// TIA Portal V16 export
// export: Created 2021-12-01T20:35:58.3632471Z, ExportSetting WithDefaults, DisplayName Totally Integrated Automation Portal, DisplayVersion V16 Update 4, DisplayName TIA Portal Version Control Interface, DisplayVersion V16 Update 2, DisplayName TIA Portal Openness, DisplayVersion V16 Update 4, DisplayName SINAMICS Startdrive Advanced, DisplayVersion V16 Update 5, DisplayName SINAMICS Startdrive G130, G150, S120, S150, SINAMICS MV, S210, DisplayVersion V16 Update 5, DisplayName SINAMICS Startdrive G110M, G120, G120C, G120D, G120P, G115D, DisplayVersion V16 Update 5, DisplayName STEP 7 Professional, DisplayVersion V16 Update 4, DisplayName STEP 7 Safety, DisplayVersion V16, DisplayName WinCC Advanced, DisplayVersion V16 Update 4
FUNCTION "ST00325_FC" : Void   // FC100, LAD
TITLE = ST00325
{ S7_Optimized_Access := 'TRUE' }
VERSION : 0.1
// stored: AutoNumber true, IsIECCheckEnabled false, SetENOAutomatically false, UDAEnableTagReadback false
   VAR_IN_OUT
      OPMODE : "OPMODE_OUT_UDT";
      HMI_EXTENSION : "HMI_EXTENSION_PANEL_UDT";
   END_VAR
   VAR_TEMP
      EmptyHS : "RT_HANDSHAKE_UDT";
      TargetSet : Bool;
      RouteSet : Bool;
      PlantIdentifier : WString;
   END_VAR
   VAR CONSTANT
      SetLocationUID : String := 'ST00325_SL';
      SetPayloadUID : String := 'ST00325_SP';
      SetAttributeUID : String := 'ST00325_SA';
   END_VAR
   VAR_TEMP   // added for the SCL form of the ladder/FBD networks
      _w1 : Bool;
      _w2 : Bool;
   END_VAR
BEGIN

REGION Network 1: Alarm
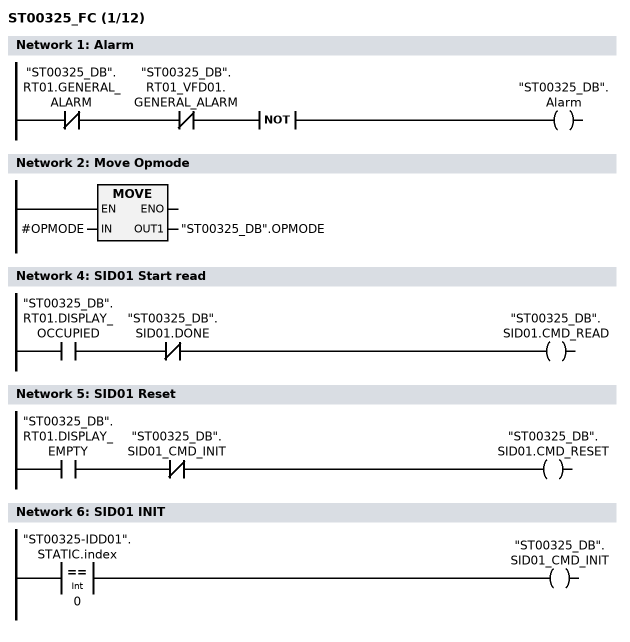
   RUNG wire#powerrail
      I_Contact( "ST00325_DB".RT01.GENERAL_ALARM )
      I_Contact( "ST00325_DB".RT01_VFD01.GENERAL_ALARM )
      Not()
      Coil( "ST00325_DB".Alarm )
   END_RUNG
   // the same network as SCL:
   "ST00325_DB".Alarm := NOT (NOT "ST00325_DB".RT01.GENERAL_ALARM AND NOT "ST00325_DB".RT01_VFD01.GENERAL_ALARM);
END_REGION

REGION Network 2: Move Opmode
   RUNG wire#powerrail
      Move(in := #OPMODE, out1 => "ST00325_DB".OPMODE)
   END_RUNG
   // the same network as SCL:
   "ST00325_DB".OPMODE := #OPMODE;
END_REGION

REGION Network 3: ==== Skid identifier Control ====
END_REGION

REGION Network 4: SID01 Start read
   RUNG wire#powerrail
      Contact( "ST00325_DB".RT01.DISPLAY_OCCUPIED )
      I_Contact( "ST00325_DB".SID01.DONE )
      Coil( "ST00325_DB".SID01.CMD_READ )
   END_RUNG
   // the same network as SCL:
   "ST00325_DB".SID01.CMD_READ := "ST00325_DB".RT01.DISPLAY_OCCUPIED AND NOT "ST00325_DB".SID01.DONE;
END_REGION

REGION Network 5: SID01 Reset
   RUNG wire#powerrail
      Contact( "ST00325_DB".RT01.DISPLAY_EMPTY )
      I_Contact( "ST00325_DB".SID01_CMD_INIT )
      Coil( "ST00325_DB".SID01.CMD_RESET )
   END_RUNG
   // the same network as SCL:
   "ST00325_DB".SID01.CMD_RESET := "ST00325_DB".RT01.DISPLAY_EMPTY AND NOT "ST00325_DB".SID01_CMD_INIT;
END_REGION

REGION Network 6: SID01 INIT
   RUNG wire#powerrail
      { S7_Templates := "SrcType := Int" } EQ_Contact(in1 := "ST00325-IDD01".STATIC.index, in2 := 0)
      Coil( "ST00325_DB".SID01_CMD_INIT )
   END_RUNG
   // the same network as SCL:
   "ST00325_DB".SID01_CMD_INIT := "ST00325-IDD01".STATIC.index = 0;
END_REGION

REGION Network 7: SID01 FB Control
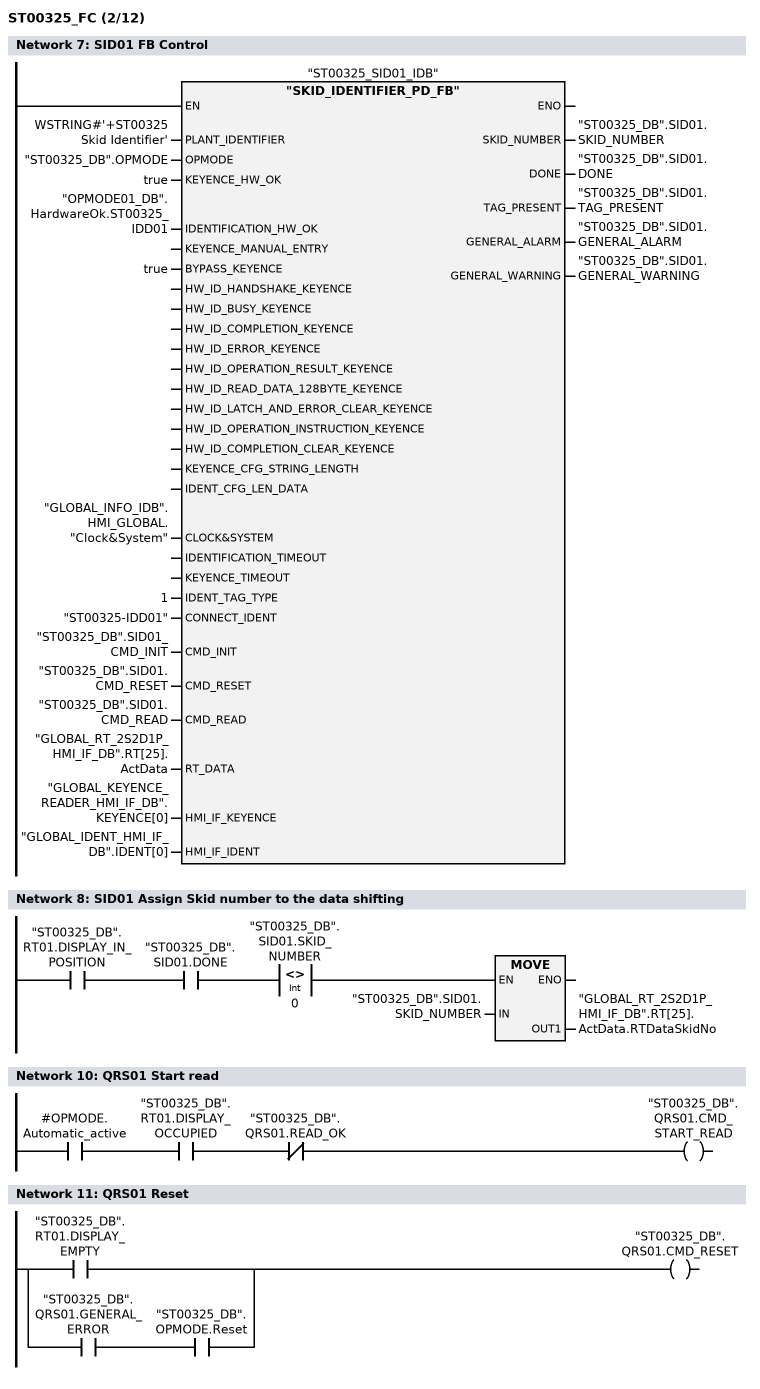
   RUNG wire#powerrail
      "ST00325_SID01_IDB"(PLANT_IDENTIFIER := WSTRING#'+ST00325 Skid Identifier', OPMODE := "ST00325_DB".OPMODE, KEYENCE_HW_OK := true, IDENTIFICATION_HW_OK := "OPMODE01_DB".HardwareOk.ST00325_IDD01, KEYENCE_MANUAL_ENTRY :=, BYPASS_KEYENCE := true, HW_ID_HANDSHAKE_KEYENCE :=, HW_ID_BUSY_KEYENCE :=, HW_ID_COMPLETION_KEYENCE :=, HW_ID_ERROR_KEYENCE :=, HW_ID_OPERATION_RESULT_KEYENCE :=, HW_ID_READ_DATA_128BYTE_KEYENCE :=, HW_ID_LATCH_AND_ERROR_CLEAR_KEYENCE :=, HW_ID_OPERATION_INSTRUCTION_KEYENCE :=, HW_ID_COMPLETION_CLEAR_KEYENCE :=, KEYENCE_CFG_STRING_LENGTH :=, IDENT_CFG_LEN_DATA :=, "CLOCK&SYSTEM" := "GLOBAL_INFO_IDB".HMI_GLOBAL."Clock&System", IDENTIFICATION_TIMEOUT :=, KEYENCE_TIMEOUT :=, IDENT_TAG_TYPE := 1, CONNECT_IDENT := "ST00325-IDD01", CMD_INIT := "ST00325_DB".SID01_CMD_INIT, CMD_RESET := "ST00325_DB".SID01.CMD_RESET, CMD_READ := "ST00325_DB".SID01.CMD_READ, RT_DATA := "GLOBAL_RT_2S2D1P_HMI_IF_DB".RT[25].ActData, HMI_IF_KEYENCE := "GLOBAL_KEYENCE_READER_HMI_IF_DB".KEYENCE[0], HMI_IF_IDENT := "GLOBAL_IDENT_HMI_IF_DB".IDENT[0], SKID_NUMBER => "ST00325_DB".SID01.SKID_NUMBER, DONE => "ST00325_DB".SID01.DONE, TAG_PRESENT => "ST00325_DB".SID01.TAG_PRESENT, GENERAL_ALARM => "ST00325_DB".SID01.GENERAL_ALARM, GENERAL_WARNING => "ST00325_DB".SID01.GENERAL_WARNING)
   END_RUNG
   // the same network as SCL:
   "ST00325_SID01_IDB"(PLANT_IDENTIFIER := WSTRING#'+ST00325 Skid Identifier',   // "SKID_IDENTIFIER_PD_FB"
                       OPMODE := "ST00325_DB".OPMODE,
                       KEYENCE_HW_OK := true,
                       IDENTIFICATION_HW_OK := "OPMODE01_DB".HardwareOk.ST00325_IDD01,
                       BYPASS_KEYENCE := true,
                       "CLOCK&SYSTEM" := "GLOBAL_INFO_IDB".HMI_GLOBAL."Clock&System",
                       IDENT_TAG_TYPE := 1,
                       CONNECT_IDENT := "ST00325-IDD01",
                       CMD_INIT := "ST00325_DB".SID01_CMD_INIT,
                       CMD_RESET := "ST00325_DB".SID01.CMD_RESET,
                       CMD_READ := "ST00325_DB".SID01.CMD_READ,
                       RT_DATA := "GLOBAL_RT_2S2D1P_HMI_IF_DB".RT[25].ActData,
                       HMI_IF_KEYENCE := "GLOBAL_KEYENCE_READER_HMI_IF_DB".KEYENCE[0],
                       HMI_IF_IDENT := "GLOBAL_IDENT_HMI_IF_DB".IDENT[0],
                       SKID_NUMBER => "ST00325_DB".SID01.SKID_NUMBER,
                       DONE => "ST00325_DB".SID01.DONE,
                       TAG_PRESENT => "ST00325_DB".SID01.TAG_PRESENT,
                       GENERAL_ALARM => "ST00325_DB".SID01.GENERAL_ALARM,
                       GENERAL_WARNING => "ST00325_DB".SID01.GENERAL_WARNING);
END_REGION

REGION Network 8: SID01 Assign Skid number to the data shifting
   RUNG wire#powerrail
      Contact( "ST00325_DB".RT01.DISPLAY_IN_POSITION )
      Contact( "ST00325_DB".SID01.DONE )
      { S7_Templates := "SrcType := Int" } NE_Contact(in1 := "ST00325_DB".SID01.SKID_NUMBER, in2 := 0)
      Move(in := "ST00325_DB".SID01.SKID_NUMBER, out1 => "GLOBAL_RT_2S2D1P_HMI_IF_DB".RT[25].ActData.RTDataSkidNo)
   END_RUNG
   // the same network as SCL:
   IF "ST00325_DB".RT01.DISPLAY_IN_POSITION AND "ST00325_DB".SID01.DONE AND ("ST00325_DB".SID01.SKID_NUMBER <> 0) THEN
       "GLOBAL_RT_2S2D1P_HMI_IF_DB".RT[25].ActData.RTDataSkidNo := "ST00325_DB".SID01.SKID_NUMBER;
   END_IF;
END_REGION

REGION Network 9: ==== Camera control ====
END_REGION

REGION Network 10: QRS01 Start read
   RUNG wire#powerrail
      Contact( #OPMODE.Automatic_active )
      Contact( "ST00325_DB".RT01.DISPLAY_OCCUPIED )
      I_Contact( "ST00325_DB".QRS01.READ_OK )
      Coil( "ST00325_DB".QRS01.CMD_START_READ )
   END_RUNG
   // the same network as SCL:
   "ST00325_DB".QRS01.CMD_START_READ := #OPMODE.Automatic_active AND "ST00325_DB".RT01.DISPLAY_OCCUPIED AND NOT "ST00325_DB".QRS01.READ_OK;
END_REGION

REGION Network 11: QRS01 Reset
   RUNG wire#powerrail
      Contact( "ST00325_DB".RT01.DISPLAY_EMPTY )
      wire#w1
      Coil( "ST00325_DB".QRS01.CMD_RESET )
   END_RUNG
   RUNG wire#powerrail
      Contact( "ST00325_DB".QRS01.GENERAL_ERROR )
      Contact( "ST00325_DB".OPMODE.Reset )
   END_RUNG wire#w1
   // the same network as SCL:
   "ST00325_DB".QRS01.CMD_RESET := "ST00325_DB".RT01.DISPLAY_EMPTY OR ("ST00325_DB".QRS01.GENERAL_ERROR AND "ST00325_DB".OPMODE.Reset);
END_REGION

REGION Network 12: QRS01 FB Control
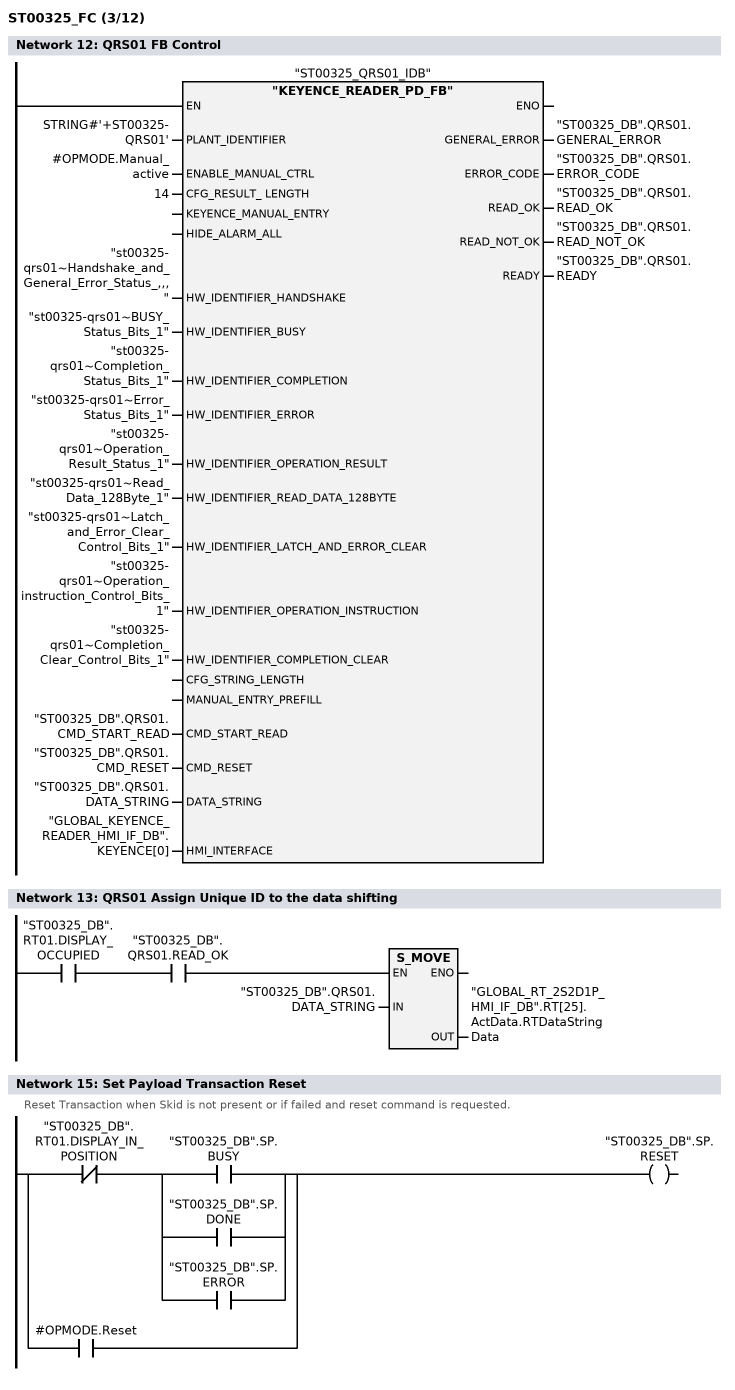
   RUNG wire#powerrail
      "ST00325_QRS01_IDB"(PLANT_IDENTIFIER := STRING#'+ST00325-QRS01', ENABLE_MANUAL_CTRL := #OPMODE.Manual_active, "CFG_RESULT_ LENGTH" := 14, KEYENCE_MANUAL_ENTRY :=, HIDE_ALARM_ALL :=, HW_IDENTIFIER_HANDSHAKE := "st00325-qrs01~Handshake_and_General_Error_Status_,,,", HW_IDENTIFIER_BUSY := "st00325-qrs01~BUSY_Status_Bits_1", HW_IDENTIFIER_COMPLETION := "st00325-qrs01~Completion_Status_Bits_1", HW_IDENTIFIER_ERROR := "st00325-qrs01~Error_Status_Bits_1", HW_IDENTIFIER_OPERATION_RESULT := "st00325-qrs01~Operation_Result_Status_1", HW_IDENTIFIER_READ_DATA_128BYTE := "st00325-qrs01~Read_Data_128Byte_1", HW_IDENTIFIER_LATCH_AND_ERROR_CLEAR := "st00325-qrs01~Latch_and_Error_Clear_Control_Bits_1", HW_IDENTIFIER_OPERATION_INSTRUCTION := "st00325-qrs01~Operation_instruction_Control_Bits_1", HW_IDENTIFIER_COMPLETION_CLEAR := "st00325-qrs01~Completion_Clear_Control_Bits_1", CFG_STRING_LENGTH :=, MANUAL_ENTRY_PREFILL :=, CMD_START_READ := "ST00325_DB".QRS01.CMD_START_READ, CMD_RESET := "ST00325_DB".QRS01.CMD_RESET, DATA_STRING := "ST00325_DB".QRS01.DATA_STRING, HMI_INTERFACE := "GLOBAL_KEYENCE_READER_HMI_IF_DB".KEYENCE[0], GENERAL_ERROR => "ST00325_DB".QRS01.GENERAL_ERROR, ERROR_CODE => "ST00325_DB".QRS01.ERROR_CODE, READ_OK => "ST00325_DB".QRS01.READ_OK, READ_NOT_OK => "ST00325_DB".QRS01.READ_NOT_OK, READY => "ST00325_DB".QRS01.READY)
   END_RUNG
   // the same network as SCL:
   "ST00325_QRS01_IDB"(PLANT_IDENTIFIER := STRING#'+ST00325-QRS01',   // "KEYENCE_READER_PD_FB"
                       ENABLE_MANUAL_CTRL := #OPMODE.Manual_active,
                       "CFG_RESULT_ LENGTH" := 14,
                       HW_IDENTIFIER_HANDSHAKE := "st00325-qrs01~Handshake_and_General_Error_Status_,,,",
                       HW_IDENTIFIER_BUSY := "st00325-qrs01~BUSY_Status_Bits_1",
                       HW_IDENTIFIER_COMPLETION := "st00325-qrs01~Completion_Status_Bits_1",
                       HW_IDENTIFIER_ERROR := "st00325-qrs01~Error_Status_Bits_1",
                       HW_IDENTIFIER_OPERATION_RESULT := "st00325-qrs01~Operation_Result_Status_1",
                       HW_IDENTIFIER_READ_DATA_128BYTE := "st00325-qrs01~Read_Data_128Byte_1",
                       HW_IDENTIFIER_LATCH_AND_ERROR_CLEAR := "st00325-qrs01~Latch_and_Error_Clear_Control_Bits_1",
                       HW_IDENTIFIER_OPERATION_INSTRUCTION := "st00325-qrs01~Operation_instruction_Control_Bits_1",
                       HW_IDENTIFIER_COMPLETION_CLEAR := "st00325-qrs01~Completion_Clear_Control_Bits_1",
                       CMD_START_READ := "ST00325_DB".QRS01.CMD_START_READ,
                       CMD_RESET := "ST00325_DB".QRS01.CMD_RESET,
                       DATA_STRING := "ST00325_DB".QRS01.DATA_STRING,
                       HMI_INTERFACE := "GLOBAL_KEYENCE_READER_HMI_IF_DB".KEYENCE[0],
                       GENERAL_ERROR => "ST00325_DB".QRS01.GENERAL_ERROR,
                       ERROR_CODE => "ST00325_DB".QRS01.ERROR_CODE,
                       READ_OK => "ST00325_DB".QRS01.READ_OK,
                       READ_NOT_OK => "ST00325_DB".QRS01.READ_NOT_OK,
                       READY => "ST00325_DB".QRS01.READY);
END_REGION

REGION Network 13: QRS01 Assign Unique ID to the data shifting
   RUNG wire#powerrail
      Contact( "ST00325_DB".RT01.DISPLAY_OCCUPIED )
      Contact( "ST00325_DB".QRS01.READ_OK )
      S_Move(in := "ST00325_DB".QRS01.DATA_STRING, out => "GLOBAL_RT_2S2D1P_HMI_IF_DB".RT[25].ActData.RTDataStringData)
   END_RUNG
   // the same network as SCL:
   IF "ST00325_DB".RT01.DISPLAY_OCCUPIED AND "ST00325_DB".QRS01.READ_OK THEN
       "GLOBAL_RT_2S2D1P_HMI_IF_DB".RT[25].ActData.RTDataStringData := "ST00325_DB".QRS01.DATA_STRING;
   END_IF;
END_REGION

REGION Network 14: ==== Set Payload ====
   // Set Payload is used to associate a BodyId (payload) to a skid
END_REGION

REGION Network 15: Set Payload Transaction Reset
   // Reset Transaction when Skid is not present or if failed and reset command is requested.
   RUNG wire#powerrail
      I_Contact( "ST00325_DB".RT01.DISPLAY_IN_POSITION )
      wire#w1
      Contact( "ST00325_DB".SP.BUSY )
      wire#w2
      Coil( "ST00325_DB".SP.RESET )
   END_RUNG
   RUNG wire#w1
      Contact( "ST00325_DB".SP.DONE )
   END_RUNG wire#w2
   RUNG wire#w1
      Contact( "ST00325_DB".SP.ERROR )
   END_RUNG wire#w2
   RUNG wire#powerrail
      Contact( #OPMODE.Reset )
   END_RUNG wire#w2
   // the same network as SCL:
   "ST00325_DB".SP.RESET := (NOT "ST00325_DB".RT01.DISPLAY_IN_POSITION AND ("ST00325_DB".SP.BUSY OR "ST00325_DB".SP.DONE OR "ST00325_DB".SP.ERROR)) OR #OPMODE.Reset;
END_REGION

REGION Network 16: Set Payload Transaction Execute
   // Execute Transaction when Skid is present and Skid Number has been retrieved.
   // Prevent further executions if transaction is in progress or has already completed.
   // 
   // To do:
   // - Remove temporary block
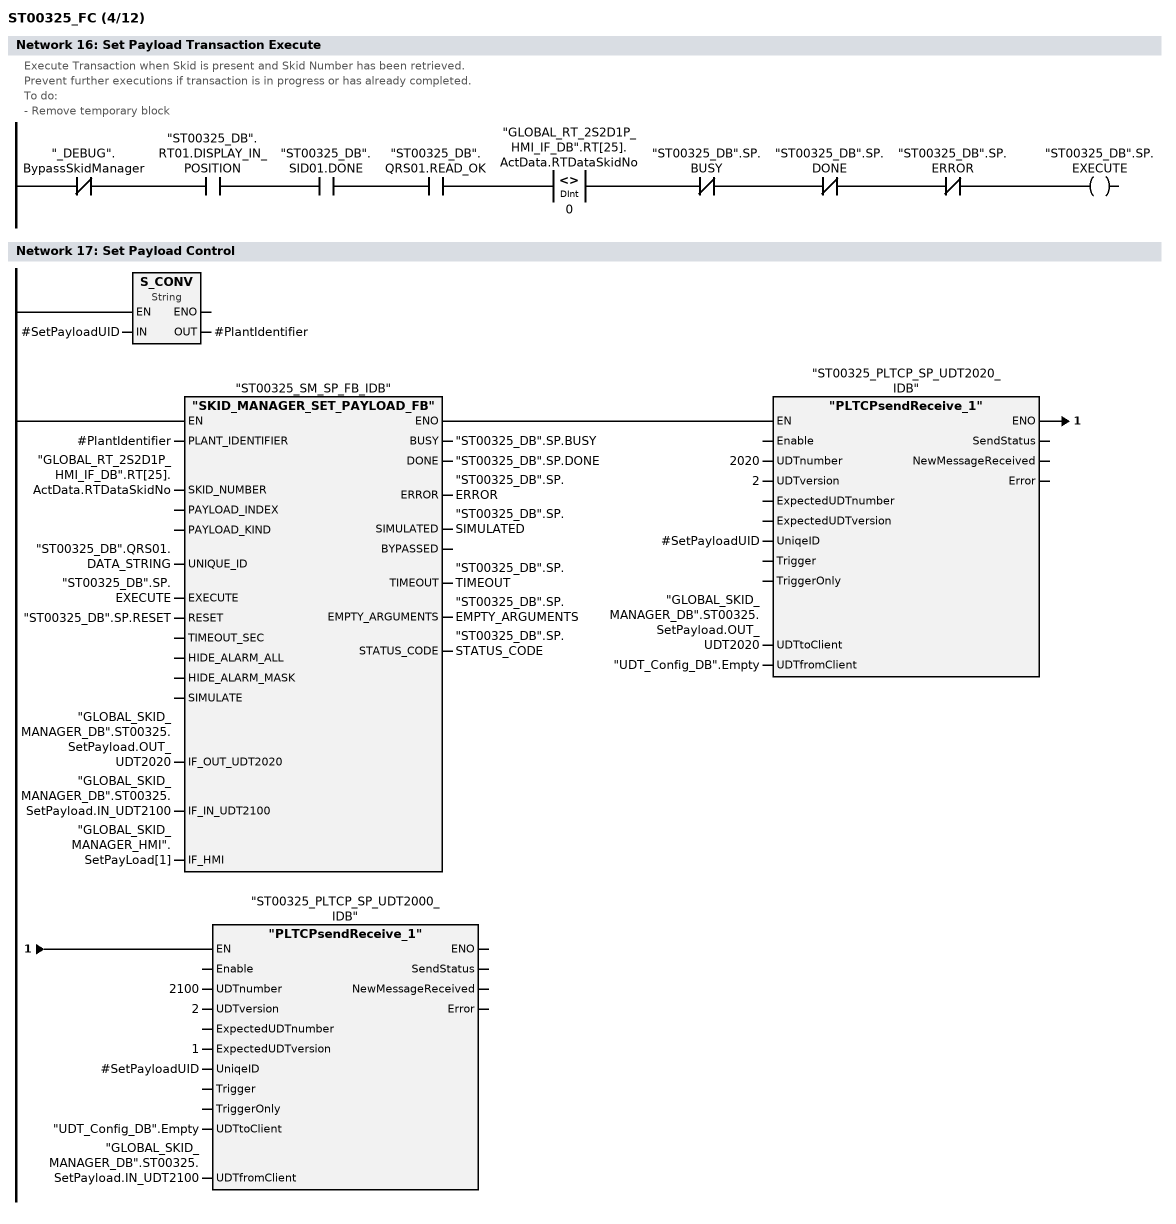
   RUNG wire#powerrail
      I_Contact( "_DEBUG".BypassSkidManager )
      Contact( "ST00325_DB".RT01.DISPLAY_IN_POSITION )
      Contact( "ST00325_DB".SID01.DONE )
      Contact( "ST00325_DB".QRS01.READ_OK )
      { S7_Templates := "SrcType := DInt" } NE_Contact(in1 := "GLOBAL_RT_2S2D1P_HMI_IF_DB".RT[25].ActData.RTDataSkidNo, in2 := 0)
      I_Contact( "ST00325_DB".SP.BUSY )
      I_Contact( "ST00325_DB".SP.DONE )
      I_Contact( "ST00325_DB".SP.ERROR )
      Coil( "ST00325_DB".SP.EXECUTE )
   END_RUNG
   // the same network as SCL:
   "ST00325_DB".SP.EXECUTE := NOT "_DEBUG".BypassSkidManager AND "ST00325_DB".RT01.DISPLAY_IN_POSITION AND "ST00325_DB".SID01.DONE AND "ST00325_DB".QRS01.READ_OK AND ("GLOBAL_RT_2S2D1P_HMI_IF_DB".RT[25].ActData.RTDataSkidNo <> 0) AND NOT "ST00325_DB".SP.BUSY AND NOT "ST00325_DB".SP.DONE AND NOT "ST00325_DB".SP.ERROR;
END_REGION

REGION Network 17: Set Payload Control
   RUNG wire#powerrail
      { S7_Templates := "[src_type := String, dest_type := WString]" } S_CONV(IN := #SetPayloadUID, OUT => #PlantIdentifier)
   END_RUNG
   RUNG wire#powerrail
      "ST00325_SM_SP_FB_IDB"(PLANT_IDENTIFIER := #PlantIdentifier, SKID_NUMBER := "GLOBAL_RT_2S2D1P_HMI_IF_DB".RT[25].ActData.RTDataSkidNo, PAYLOAD_INDEX :=, PAYLOAD_KIND :=, UNIQUE_ID := "ST00325_DB".QRS01.DATA_STRING, EXECUTE := "ST00325_DB".SP.EXECUTE, RESET := "ST00325_DB".SP.RESET, TIMEOUT_SEC :=, HIDE_ALARM_ALL :=, HIDE_ALARM_MASK :=, SIMULATE :=, IF_OUT_UDT2020 := "GLOBAL_SKID_MANAGER_DB".ST00325.SetPayload.OUT_UDT2020, IF_IN_UDT2100 := "GLOBAL_SKID_MANAGER_DB".ST00325.SetPayload.IN_UDT2100, IF_HMI := "GLOBAL_SKID_MANAGER_HMI".SetPayLoad[1], BUSY => "ST00325_DB".SP.BUSY, DONE => "ST00325_DB".SP.DONE, ERROR => "ST00325_DB".SP.ERROR, SIMULATED => "ST00325_DB".SP.SIMULATED, BYPASSED =>, TIMEOUT => "ST00325_DB".SP.TIMEOUT, EMPTY_ARGUMENTS => "ST00325_DB".SP.EMPTY_ARGUMENTS, STATUS_CODE => "ST00325_DB".SP.STATUS_CODE)
      "ST00325_PLTCP_SP_UDT2020_IDB"(Enable :=, UDTnumber := 2020, UDTversion := 2, ExpectedUDTnumber :=, ExpectedUDTversion :=, UniqeID := #SetPayloadUID, Trigger :=, TriggerOnly :=, UDTtoClient := "GLOBAL_SKID_MANAGER_DB".ST00325.SetPayload.OUT_UDT2020, UDTfromClient := "UDT_Config_DB".Empty, SendStatus =>, NewMessageReceived =>, Error =>)
      "ST00325_PLTCP_SP_UDT2000_IDB"(Enable :=, UDTnumber := 2100, UDTversion := 2, ExpectedUDTnumber :=, ExpectedUDTversion := 1, UniqeID := #SetPayloadUID, Trigger :=, TriggerOnly :=, UDTtoClient := "UDT_Config_DB".Empty, UDTfromClient := "GLOBAL_SKID_MANAGER_DB".ST00325.SetPayload.IN_UDT2100, SendStatus =>, NewMessageReceived =>, Error =>)
   END_RUNG
   // the same network as SCL:
   S_CONV(IN := #SetPayloadUID, OUT => #PlantIdentifier);
   "ST00325_SM_SP_FB_IDB"(PLANT_IDENTIFIER := #PlantIdentifier,   // "SKID_MANAGER_SET_PAYLOAD_FB"
                          SKID_NUMBER := "GLOBAL_RT_2S2D1P_HMI_IF_DB".RT[25].ActData.RTDataSkidNo,
                          UNIQUE_ID := "ST00325_DB".QRS01.DATA_STRING,
                          EXECUTE := "ST00325_DB".SP.EXECUTE,
                          RESET := "ST00325_DB".SP.RESET,
                          IF_OUT_UDT2020 := "GLOBAL_SKID_MANAGER_DB".ST00325.SetPayload.OUT_UDT2020,
                          IF_IN_UDT2100 := "GLOBAL_SKID_MANAGER_DB".ST00325.SetPayload.IN_UDT2100,
                          IF_HMI := "GLOBAL_SKID_MANAGER_HMI".SetPayLoad[1],
                          BUSY => "ST00325_DB".SP.BUSY,
                          DONE => "ST00325_DB".SP.DONE,
                          ERROR => "ST00325_DB".SP.ERROR,
                          SIMULATED => "ST00325_DB".SP.SIMULATED,
                          TIMEOUT => "ST00325_DB".SP.TIMEOUT,
                          EMPTY_ARGUMENTS => "ST00325_DB".SP.EMPTY_ARGUMENTS,
                          STATUS_CODE => "ST00325_DB".SP.STATUS_CODE,
                          ENO => #_w1);
   "ST00325_PLTCP_SP_UDT2020_IDB"(EN := #_w1,   // "PLTCPsendReceive_1"
                           UDTnumber := 2020,
                           UDTversion := 2,
                           UniqeID := #SetPayloadUID,
                           UDTtoClient := "GLOBAL_SKID_MANAGER_DB".ST00325.SetPayload.OUT_UDT2020,
                           UDTfromClient := "UDT_Config_DB".Empty,
                           ENO => #_w2);
   IF #_w2 THEN
       "ST00325_PLTCP_SP_UDT2000_IDB"(UDTnumber := 2100,   // "PLTCPsendReceive_1"
                               UDTversion := 2,
                               ExpectedUDTversion := 1,
                               UniqeID := #SetPayloadUID,
                               UDTtoClient := "UDT_Config_DB".Empty,
                               UDTfromClient := "GLOBAL_SKID_MANAGER_DB".ST00325.SetPayload.IN_UDT2100);
   END_IF;
END_REGION

REGION Network 18: ==== Set Location ====
END_REGION

REGION Network 19: Set Location Transaction Reset
   // Reset Transaction when Skid is not present or if failed and reset command is requested.
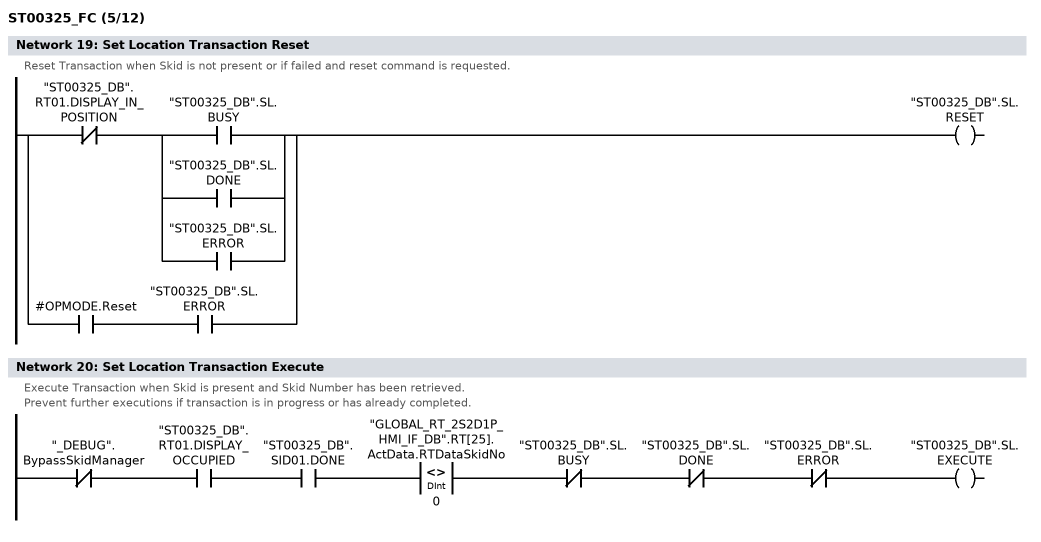
   RUNG wire#powerrail
      I_Contact( "ST00325_DB".RT01.DISPLAY_IN_POSITION )
      wire#w1
      Contact( "ST00325_DB".SL.BUSY )
      wire#w2
      Coil( "ST00325_DB".SL.RESET )
   END_RUNG
   RUNG wire#w1
      Contact( "ST00325_DB".SL.DONE )
   END_RUNG wire#w2
   RUNG wire#w1
      Contact( "ST00325_DB".SL.ERROR )
   END_RUNG wire#w2
   RUNG wire#powerrail
      Contact( #OPMODE.Reset )
      Contact( "ST00325_DB".SL.ERROR )
   END_RUNG wire#w2
   // the same network as SCL:
   "ST00325_DB".SL.RESET := (NOT "ST00325_DB".RT01.DISPLAY_IN_POSITION AND ("ST00325_DB".SL.BUSY OR "ST00325_DB".SL.DONE OR "ST00325_DB".SL.ERROR)) OR (#OPMODE.Reset AND "ST00325_DB".SL.ERROR);
END_REGION

REGION Network 20: Set Location Transaction Execute
   // Execute Transaction when Skid is present and Skid Number has been retrieved.
   // Prevent further executions if transaction is in progress or has already completed.
   RUNG wire#powerrail
      I_Contact( "_DEBUG".BypassSkidManager )
      Contact( "ST00325_DB".RT01.DISPLAY_OCCUPIED )
      Contact( "ST00325_DB".SID01.DONE )
      { S7_Templates := "SrcType := DInt" } NE_Contact(in1 := "GLOBAL_RT_2S2D1P_HMI_IF_DB".RT[25].ActData.RTDataSkidNo, in2 := 0)
      I_Contact( "ST00325_DB".SL.BUSY )
      I_Contact( "ST00325_DB".SL.DONE )
      I_Contact( "ST00325_DB".SL.ERROR )
      Coil( "ST00325_DB".SL.EXECUTE )
   END_RUNG
   // the same network as SCL:
   "ST00325_DB".SL.EXECUTE := NOT "_DEBUG".BypassSkidManager AND "ST00325_DB".RT01.DISPLAY_OCCUPIED AND "ST00325_DB".SID01.DONE AND ("GLOBAL_RT_2S2D1P_HMI_IF_DB".RT[25].ActData.RTDataSkidNo <> 0) AND NOT "ST00325_DB".SL.BUSY AND NOT "ST00325_DB".SL.DONE AND NOT "ST00325_DB".SL.ERROR;
END_REGION

REGION Network 21: Set Location Control
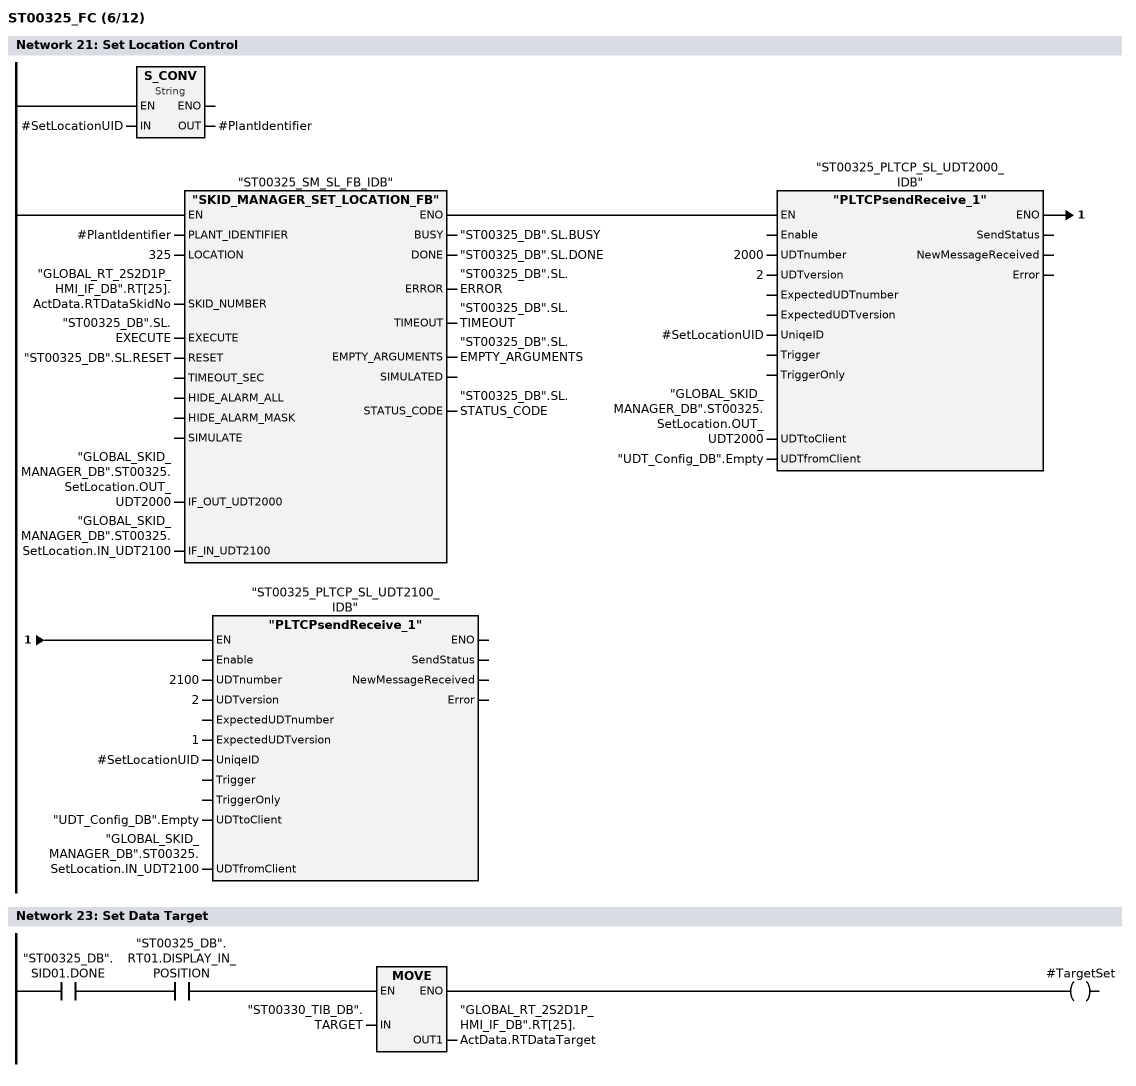
   RUNG wire#powerrail
      { S7_Templates := "[src_type := String, dest_type := WString]" } S_CONV(IN := #SetLocationUID, OUT => #PlantIdentifier)
   END_RUNG
   RUNG wire#powerrail
      "ST00325_SM_SL_FB_IDB"(PLANT_IDENTIFIER := #PlantIdentifier, LOCATION := 325, SKID_NUMBER := "GLOBAL_RT_2S2D1P_HMI_IF_DB".RT[25].ActData.RTDataSkidNo, EXECUTE := "ST00325_DB".SL.EXECUTE, RESET := "ST00325_DB".SL.RESET, TIMEOUT_SEC :=, HIDE_ALARM_ALL :=, HIDE_ALARM_MASK :=, SIMULATE :=, IF_OUT_UDT2000 := "GLOBAL_SKID_MANAGER_DB".ST00325.SetLocation.OUT_UDT2000, IF_IN_UDT2100 := "GLOBAL_SKID_MANAGER_DB".ST00325.SetLocation.IN_UDT2100, BUSY => "ST00325_DB".SL.BUSY, DONE => "ST00325_DB".SL.DONE, ERROR => "ST00325_DB".SL.ERROR, TIMEOUT => "ST00325_DB".SL.TIMEOUT, EMPTY_ARGUMENTS => "ST00325_DB".SL.EMPTY_ARGUMENTS, SIMULATED =>, STATUS_CODE => "ST00325_DB".SL.STATUS_CODE)
      "ST00325_PLTCP_SL_UDT2000_IDB"(Enable :=, UDTnumber := 2000, UDTversion := 2, ExpectedUDTnumber :=, ExpectedUDTversion :=, UniqeID := #SetLocationUID, Trigger :=, TriggerOnly :=, UDTtoClient := "GLOBAL_SKID_MANAGER_DB".ST00325.SetLocation.OUT_UDT2000, UDTfromClient := "UDT_Config_DB".Empty, SendStatus =>, NewMessageReceived =>, Error =>)
      "ST00325_PLTCP_SL_UDT2100_IDB"(Enable :=, UDTnumber := 2100, UDTversion := 2, ExpectedUDTnumber :=, ExpectedUDTversion := 1, UniqeID := #SetLocationUID, Trigger :=, TriggerOnly :=, UDTtoClient := "UDT_Config_DB".Empty, UDTfromClient := "GLOBAL_SKID_MANAGER_DB".ST00325.SetLocation.IN_UDT2100, SendStatus =>, NewMessageReceived =>, Error =>)
   END_RUNG
   // the same network as SCL:
   S_CONV(IN := #SetLocationUID, OUT => #PlantIdentifier);
   "ST00325_SM_SL_FB_IDB"(PLANT_IDENTIFIER := #PlantIdentifier,   // "SKID_MANAGER_SET_LOCATION_FB"
                          LOCATION := 325,
                          SKID_NUMBER := "GLOBAL_RT_2S2D1P_HMI_IF_DB".RT[25].ActData.RTDataSkidNo,
                          EXECUTE := "ST00325_DB".SL.EXECUTE,
                          RESET := "ST00325_DB".SL.RESET,
                          IF_OUT_UDT2000 := "GLOBAL_SKID_MANAGER_DB".ST00325.SetLocation.OUT_UDT2000,
                          IF_IN_UDT2100 := "GLOBAL_SKID_MANAGER_DB".ST00325.SetLocation.IN_UDT2100,
                          BUSY => "ST00325_DB".SL.BUSY,
                          DONE => "ST00325_DB".SL.DONE,
                          ERROR => "ST00325_DB".SL.ERROR,
                          TIMEOUT => "ST00325_DB".SL.TIMEOUT,
                          EMPTY_ARGUMENTS => "ST00325_DB".SL.EMPTY_ARGUMENTS,
                          STATUS_CODE => "ST00325_DB".SL.STATUS_CODE,
                          ENO => #_w1);
   "ST00325_PLTCP_SL_UDT2000_IDB"(EN := #_w1,   // "PLTCPsendReceive_1"
                           UDTnumber := 2000,
                           UDTversion := 2,
                           UniqeID := #SetLocationUID,
                           UDTtoClient := "GLOBAL_SKID_MANAGER_DB".ST00325.SetLocation.OUT_UDT2000,
                           UDTfromClient := "UDT_Config_DB".Empty,
                           ENO => #_w2);
   IF #_w2 THEN
       "ST00325_PLTCP_SL_UDT2100_IDB"(UDTnumber := 2100,   // "PLTCPsendReceive_1"
                               UDTversion := 2,
                               ExpectedUDTversion := 1,
                               UniqeID := #SetLocationUID,
                               UDTtoClient := "UDT_Config_DB".Empty,
                               UDTfromClient := "GLOBAL_SKID_MANAGER_DB".ST00325.SetLocation.IN_UDT2100);
   END_IF;
END_REGION

REGION Network 22: ==== Routing control ====
END_REGION

REGION Network 23: Set Data Target
   RUNG wire#powerrail
      Contact( "ST00325_DB".SID01.DONE )
      Contact( "ST00325_DB".RT01.DISPLAY_IN_POSITION )
      Move(in := "ST00330_TIB_DB".TARGET, out1 => "GLOBAL_RT_2S2D1P_HMI_IF_DB".RT[25].ActData.RTDataTarget)
      Coil( #TargetSet )
   END_RUNG
   // the same network as SCL:
   #_w1 := "ST00325_DB".SID01.DONE AND "ST00325_DB".RT01.DISPLAY_IN_POSITION;
   IF #_w1 THEN "GLOBAL_RT_2S2D1P_HMI_IF_DB".RT[25].ActData.RTDataTarget := "ST00330_TIB_DB".TARGET; END_IF;
   #TargetSet := #_w1;
END_REGION

REGION Network 24: Set route
   // To do:
   // - Determine whether skid is carrying production body or doors/liftgates
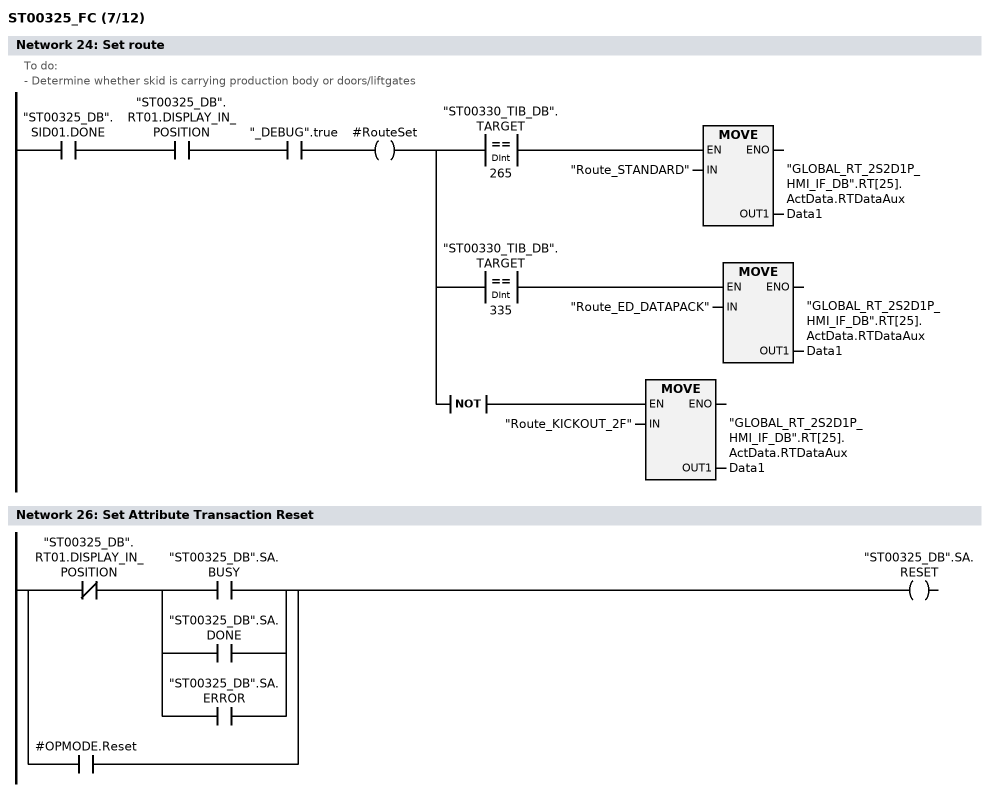
   RUNG wire#powerrail
      Contact( "ST00325_DB".SID01.DONE )
      Contact( "ST00325_DB".RT01.DISPLAY_IN_POSITION )
      Contact( "_DEBUG".true )
      Coil( #RouteSet )
      wire#w1
      { S7_Templates := "SrcType := DInt" } EQ_Contact(in1 := "ST00330_TIB_DB".TARGET, in2 := 265)
      Move(in := "Route_STANDARD", out1 => "GLOBAL_RT_2S2D1P_HMI_IF_DB".RT[25].ActData.RTDataAuxData1)
   END_RUNG
   RUNG wire#w1
      { S7_Templates := "SrcType := DInt" } EQ_Contact(in1 := "ST00330_TIB_DB".TARGET, in2 := 335)
      Move(in := "Route_ED_DATAPACK", out1 => "GLOBAL_RT_2S2D1P_HMI_IF_DB".RT[25].ActData.RTDataAuxData1)
   END_RUNG
   RUNG wire#w1
      Not()
      Move(in := "Route_KICKOUT_2F", out1 => "GLOBAL_RT_2S2D1P_HMI_IF_DB".RT[25].ActData.RTDataAuxData1)
   END_RUNG
   // the same network as SCL:
   #RouteSet := "ST00325_DB".SID01.DONE AND "ST00325_DB".RT01.DISPLAY_IN_POSITION AND "_DEBUG".true;
   IF #RouteSet AND ("ST00330_TIB_DB".TARGET = 265) THEN
       "GLOBAL_RT_2S2D1P_HMI_IF_DB".RT[25].ActData.RTDataAuxData1 := "Route_STANDARD";
   END_IF;
   IF #RouteSet AND ("ST00330_TIB_DB".TARGET = 335) THEN
       "GLOBAL_RT_2S2D1P_HMI_IF_DB".RT[25].ActData.RTDataAuxData1 := "Route_ED_DATAPACK";
   END_IF;
   IF NOT #RouteSet THEN
       "GLOBAL_RT_2S2D1P_HMI_IF_DB".RT[25].ActData.RTDataAuxData1 := "Route_KICKOUT_2F";
   END_IF;
END_REGION

REGION Network 25: ==== Set Attribute ====
END_REGION

REGION Network 26: Set Attribute Transaction Reset
   RUNG wire#powerrail
      I_Contact( "ST00325_DB".RT01.DISPLAY_IN_POSITION )
      wire#w1
      Contact( "ST00325_DB".SA.BUSY )
      wire#w2
      Coil( "ST00325_DB".SA.RESET )
   END_RUNG
   RUNG wire#w1
      Contact( "ST00325_DB".SA.DONE )
   END_RUNG wire#w2
   RUNG wire#w1
      Contact( "ST00325_DB".SA.ERROR )
   END_RUNG wire#w2
   RUNG wire#powerrail
      Contact( #OPMODE.Reset )
   END_RUNG wire#w2
   // the same network as SCL:
   "ST00325_DB".SA.RESET := (NOT "ST00325_DB".RT01.DISPLAY_IN_POSITION AND ("ST00325_DB".SA.BUSY OR "ST00325_DB".SA.DONE OR "ST00325_DB".SA.ERROR)) OR #OPMODE.Reset;
END_REGION

REGION Network 27: Set Attribute Value
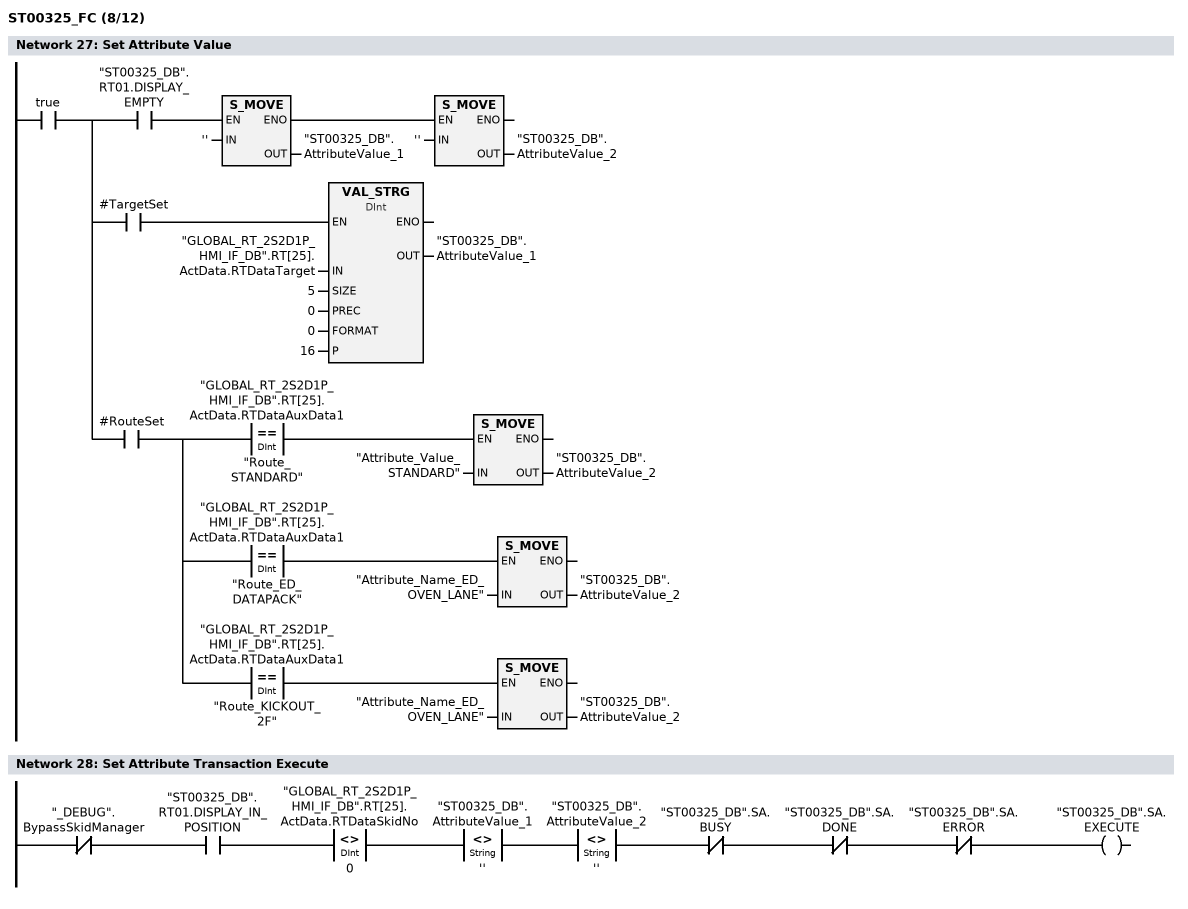
   RUNG wire#powerrail
      Contact( true )
      wire#w1
      Contact( "ST00325_DB".RT01.DISPLAY_EMPTY )
      S_Move(in := '', out => "ST00325_DB".AttributeValue_1)
      S_Move(in := '', out => "ST00325_DB".AttributeValue_2)
   END_RUNG
   RUNG wire#w1
      Contact( #TargetSet )
      { S7_Templates := "[value_type := DInt, str_type := String]" } VAL_STRG(IN := "GLOBAL_RT_2S2D1P_HMI_IF_DB".RT[25].ActData.RTDataTarget, SIZE := 5, PREC := 0, FORMAT := 0, P := 16, OUT => "ST00325_DB".AttributeValue_1)
   END_RUNG
   RUNG wire#w1
      Contact( #RouteSet )
      wire#w2
      { S7_Templates := "SrcType := DInt" } EQ_Contact(in1 := "GLOBAL_RT_2S2D1P_HMI_IF_DB".RT[25].ActData.RTDataAuxData1, in2 := "Route_STANDARD")
      S_Move(in := "Attribute_Value_STANDARD", out => "ST00325_DB".AttributeValue_2)
   END_RUNG
   RUNG wire#w2
      { S7_Templates := "SrcType := DInt" } EQ_Contact(in1 := "GLOBAL_RT_2S2D1P_HMI_IF_DB".RT[25].ActData.RTDataAuxData1, in2 := "Route_ED_DATAPACK")
      S_Move(in := "Attribute_Name_ED_OVEN_LANE", out => "ST00325_DB".AttributeValue_2)
   END_RUNG
   RUNG wire#w2
      { S7_Templates := "SrcType := DInt" } EQ_Contact(in1 := "GLOBAL_RT_2S2D1P_HMI_IF_DB".RT[25].ActData.RTDataAuxData1, in2 := "Route_KICKOUT_2F")
      S_Move(in := "Attribute_Name_ED_OVEN_LANE", out => "ST00325_DB".AttributeValue_2)
   END_RUNG
   // the same network as SCL:
   IF true AND "ST00325_DB".RT01.DISPLAY_EMPTY THEN
       "ST00325_DB".AttributeValue_1 := '';
       "ST00325_DB".AttributeValue_2 := '';
   END_IF;
   IF true AND #TargetSet THEN
       VAL_STRG(IN := "GLOBAL_RT_2S2D1P_HMI_IF_DB".RT[25].ActData.RTDataTarget,
                SIZE := 5,
                PREC := 0,
                FORMAT := 0,
                P := 16,
                OUT => "ST00325_DB".AttributeValue_1);
   END_IF;
   #_w1 := true AND #RouteSet;
   IF #_w1 AND ("GLOBAL_RT_2S2D1P_HMI_IF_DB".RT[25].ActData.RTDataAuxData1 = "Route_STANDARD") THEN
       "ST00325_DB".AttributeValue_2 := "Attribute_Value_STANDARD";
   END_IF;
   IF #_w1 AND ("GLOBAL_RT_2S2D1P_HMI_IF_DB".RT[25].ActData.RTDataAuxData1 = "Route_ED_DATAPACK") THEN
       "ST00325_DB".AttributeValue_2 := "Attribute_Name_ED_OVEN_LANE";
   END_IF;
   IF #_w1 AND ("GLOBAL_RT_2S2D1P_HMI_IF_DB".RT[25].ActData.RTDataAuxData1 = "Route_KICKOUT_2F") THEN
       "ST00325_DB".AttributeValue_2 := "Attribute_Name_ED_OVEN_LANE";
   END_IF;
END_REGION

REGION Network 28: Set Attribute Transaction Execute
   RUNG wire#powerrail
      I_Contact( "_DEBUG".BypassSkidManager )
      Contact( "ST00325_DB".RT01.DISPLAY_IN_POSITION )
      { S7_Templates := "SrcType := DInt" } NE_Contact(in1 := "GLOBAL_RT_2S2D1P_HMI_IF_DB".RT[25].ActData.RTDataSkidNo, in2 := 0)
      { S7_Templates := "SrcType := String" } NE_Contact(in1 := "ST00325_DB".AttributeValue_1, in2 := '')
      { S7_Templates := "SrcType := String" } NE_Contact(in1 := "ST00325_DB".AttributeValue_2, in2 := '')
      I_Contact( "ST00325_DB".SA.BUSY )
      I_Contact( "ST00325_DB".SA.DONE )
      I_Contact( "ST00325_DB".SA.ERROR )
      Coil( "ST00325_DB".SA.EXECUTE )
   END_RUNG
   // the same network as SCL:
   "ST00325_DB".SA.EXECUTE := NOT "_DEBUG".BypassSkidManager AND "ST00325_DB".RT01.DISPLAY_IN_POSITION AND ("GLOBAL_RT_2S2D1P_HMI_IF_DB".RT[25].ActData.RTDataSkidNo <> 0) AND ("ST00325_DB".AttributeValue_1 <> '') AND ("ST00325_DB".AttributeValue_2 <> '') AND NOT "ST00325_DB".SA.BUSY AND NOT "ST00325_DB".SA.DONE AND NOT "ST00325_DB".SA.ERROR;
END_REGION

REGION Network 29: Set Attribute Transaction Control
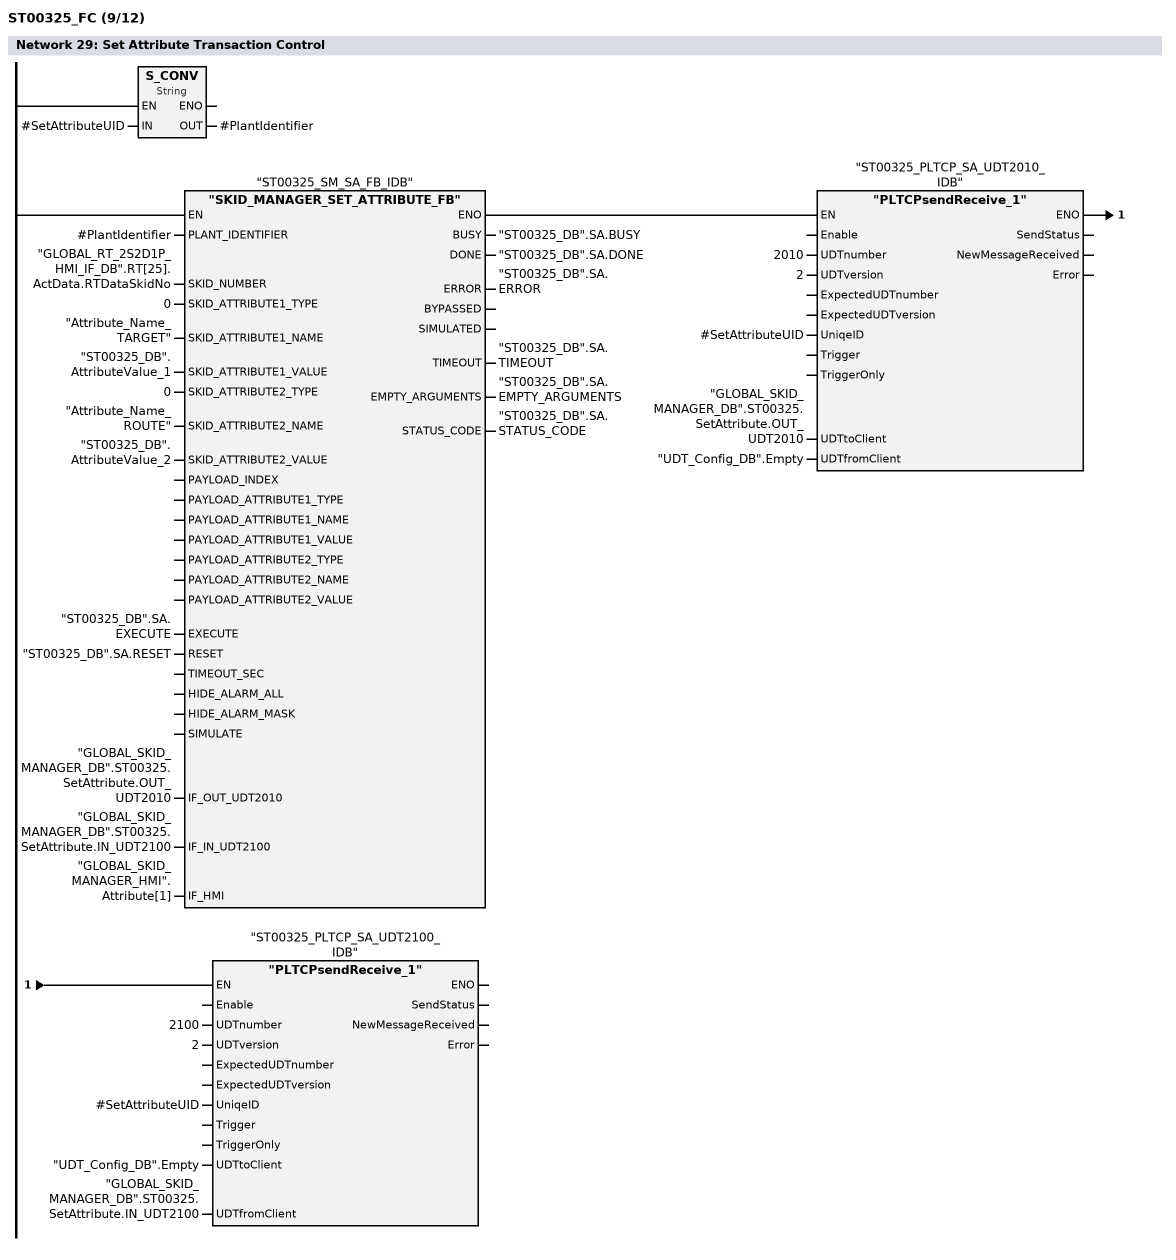
   RUNG wire#powerrail
      { S7_Templates := "[src_type := String, dest_type := WString]" } S_CONV(IN := #SetAttributeUID, OUT => #PlantIdentifier)
   END_RUNG
   RUNG wire#powerrail
      "ST00325_SM_SA_FB_IDB"(PLANT_IDENTIFIER := #PlantIdentifier, SKID_NUMBER := "GLOBAL_RT_2S2D1P_HMI_IF_DB".RT[25].ActData.RTDataSkidNo, SKID_ATTRIBUTE1_TYPE := 0, SKID_ATTRIBUTE1_NAME := "Attribute_Name_TARGET", SKID_ATTRIBUTE1_VALUE := "ST00325_DB".AttributeValue_1, SKID_ATTRIBUTE2_TYPE := 0, SKID_ATTRIBUTE2_NAME := "Attribute_Name_ROUTE", SKID_ATTRIBUTE2_VALUE := "ST00325_DB".AttributeValue_2, PAYLOAD_INDEX :=, PAYLOAD_ATTRIBUTE1_TYPE :=, PAYLOAD_ATTRIBUTE1_NAME :=, PAYLOAD_ATTRIBUTE1_VALUE :=, PAYLOAD_ATTRIBUTE2_TYPE :=, PAYLOAD_ATTRIBUTE2_NAME :=, PAYLOAD_ATTRIBUTE2_VALUE :=, EXECUTE := "ST00325_DB".SA.EXECUTE, RESET := "ST00325_DB".SA.RESET, TIMEOUT_SEC :=, HIDE_ALARM_ALL :=, HIDE_ALARM_MASK :=, SIMULATE :=, IF_OUT_UDT2010 := "GLOBAL_SKID_MANAGER_DB".ST00325.SetAttribute.OUT_UDT2010, IF_IN_UDT2100 := "GLOBAL_SKID_MANAGER_DB".ST00325.SetAttribute.IN_UDT2100, IF_HMI := "GLOBAL_SKID_MANAGER_HMI".Attribute[1], BUSY => "ST00325_DB".SA.BUSY, DONE => "ST00325_DB".SA.DONE, ERROR => "ST00325_DB".SA.ERROR, BYPASSED =>, SIMULATED =>, TIMEOUT => "ST00325_DB".SA.TIMEOUT, EMPTY_ARGUMENTS => "ST00325_DB".SA.EMPTY_ARGUMENTS, STATUS_CODE => "ST00325_DB".SA.STATUS_CODE)
      "ST00325_PLTCP_SA_UDT2010_IDB"(Enable :=, UDTnumber := 2010, UDTversion := 2, ExpectedUDTnumber :=, ExpectedUDTversion :=, UniqeID := #SetAttributeUID, Trigger :=, TriggerOnly :=, UDTtoClient := "GLOBAL_SKID_MANAGER_DB".ST00325.SetAttribute.OUT_UDT2010, UDTfromClient := "UDT_Config_DB".Empty, SendStatus =>, NewMessageReceived =>, Error =>)
      "ST00325_PLTCP_SA_UDT2100_IDB"(Enable :=, UDTnumber := 2100, UDTversion := 2, ExpectedUDTnumber :=, ExpectedUDTversion :=, UniqeID := #SetAttributeUID, Trigger :=, TriggerOnly :=, UDTtoClient := "UDT_Config_DB".Empty, UDTfromClient := "GLOBAL_SKID_MANAGER_DB".ST00325.SetAttribute.IN_UDT2100, SendStatus =>, NewMessageReceived =>, Error =>)
   END_RUNG
   // the same network as SCL:
   S_CONV(IN := #SetAttributeUID, OUT => #PlantIdentifier);
   "ST00325_SM_SA_FB_IDB"(PLANT_IDENTIFIER := #PlantIdentifier,   // "SKID_MANAGER_SET_ATTRIBUTE_FB"
                          SKID_NUMBER := "GLOBAL_RT_2S2D1P_HMI_IF_DB".RT[25].ActData.RTDataSkidNo,
                          SKID_ATTRIBUTE1_TYPE := 0,
                          SKID_ATTRIBUTE1_NAME := "Attribute_Name_TARGET",
                          SKID_ATTRIBUTE1_VALUE := "ST00325_DB".AttributeValue_1,
                          SKID_ATTRIBUTE2_TYPE := 0,
                          SKID_ATTRIBUTE2_NAME := "Attribute_Name_ROUTE",
                          SKID_ATTRIBUTE2_VALUE := "ST00325_DB".AttributeValue_2,
                          EXECUTE := "ST00325_DB".SA.EXECUTE,
                          RESET := "ST00325_DB".SA.RESET,
                          IF_OUT_UDT2010 := "GLOBAL_SKID_MANAGER_DB".ST00325.SetAttribute.OUT_UDT2010,
                          IF_IN_UDT2100 := "GLOBAL_SKID_MANAGER_DB".ST00325.SetAttribute.IN_UDT2100,
                          IF_HMI := "GLOBAL_SKID_MANAGER_HMI".Attribute[1],
                          BUSY => "ST00325_DB".SA.BUSY,
                          DONE => "ST00325_DB".SA.DONE,
                          ERROR => "ST00325_DB".SA.ERROR,
                          TIMEOUT => "ST00325_DB".SA.TIMEOUT,
                          EMPTY_ARGUMENTS => "ST00325_DB".SA.EMPTY_ARGUMENTS,
                          STATUS_CODE => "ST00325_DB".SA.STATUS_CODE,
                          ENO => #_w1);
   "ST00325_PLTCP_SA_UDT2010_IDB"(EN := #_w1,   // "PLTCPsendReceive_1"
                           UDTnumber := 2010,
                           UDTversion := 2,
                           UniqeID := #SetAttributeUID,
                           UDTtoClient := "GLOBAL_SKID_MANAGER_DB".ST00325.SetAttribute.OUT_UDT2010,
                           UDTfromClient := "UDT_Config_DB".Empty,
                           ENO => #_w2);
   IF #_w2 THEN
       "ST00325_PLTCP_SA_UDT2100_IDB"(UDTnumber := 2100,   // "PLTCPsendReceive_1"
                               UDTversion := 2,
                               UniqeID := #SetAttributeUID,
                               UDTtoClient := "UDT_Config_DB".Empty,
                               UDTfromClient := "GLOBAL_SKID_MANAGER_DB".ST00325.SetAttribute.IN_UDT2100);
   END_IF;
END_REGION

REGION Network 30: *******************RT01 Control*******************
END_REGION

REGION Network 31 (SCL): RT01 Parameters
   "ST00325_DB".RT01.PARA_SET.Para.PosEndForward1 := true;
   "ST00325_DB".RT01.PARA_SET.Para.PosEndReverse := true;
   "ST00325_DB".RT01.PARA_SET.Para.PosSlowForward := true;

   "ST00325_DB".RT01.PARA_SET.Set.RunTimeForward := 600;
   "ST00325_DB".RT01.PARA_SET.Set.RunTimeReverse := 450;
   "ST00325_DB".RT01.PARA_SET.Set.DelayPosReverse := 0;
END_REGION

REGION Network 32: RT01 HandShake
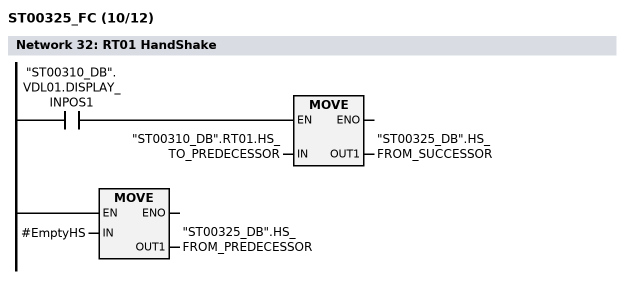
   RUNG wire#powerrail
      Contact( "ST00310_DB".VDL01.DISPLAY_INPOS1 )
      Move(in := "ST00310_DB".RT01.HS_TO_PREDECESSOR, out1 => "ST00325_DB".HS_FROM_SUCCESSOR)
   END_RUNG
   RUNG wire#powerrail
      Move(in := #EmptyHS, out1 => "ST00325_DB".HS_FROM_PREDECESSOR)
   END_RUNG
   // the same network as SCL:
   IF "ST00310_DB".VDL01.DISPLAY_INPOS1 THEN
       "ST00325_DB".HS_FROM_SUCCESSOR := "ST00310_DB".RT01.HS_TO_PREDECESSOR;
   END_IF;
   "ST00325_DB".HS_FROM_PREDECESSOR := #EmptyHS;
END_REGION

REGION Network 33: RT01 FB Control
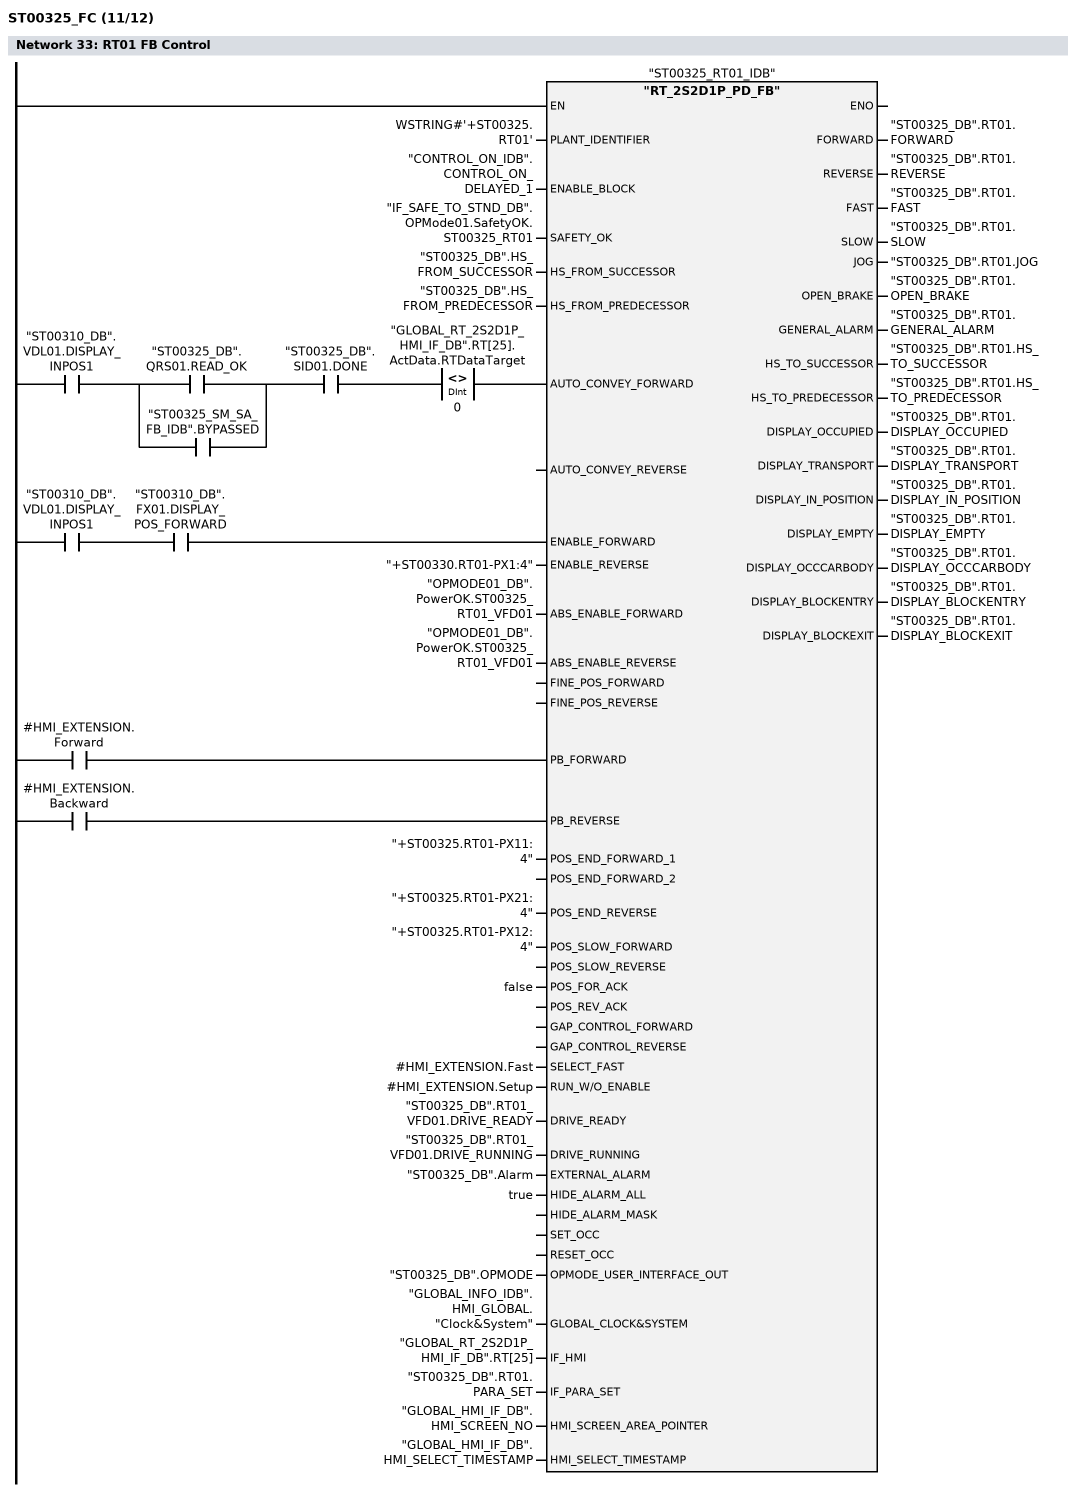
   RUNG wire#powerrail
      "ST00325_RT01_IDB"(AUTO_CONVEY_FORWARD := wire#w3, ENABLE_FORWARD := wire#w4, PB_FORWARD := wire#w5, PB_REVERSE := wire#w6, PLANT_IDENTIFIER := WSTRING#'+ST00325.RT01', ENABLE_BLOCK := "CONTROL_ON_IDB".CONTROL_ON_DELAYED_1, SAFETY_OK := "IF_SAFE_TO_STND_DB".OPMode01.SafetyOK.ST00325_RT01, HS_FROM_SUCCESSOR := "ST00325_DB".HS_FROM_SUCCESSOR, HS_FROM_PREDECESSOR := "ST00325_DB".HS_FROM_PREDECESSOR, AUTO_CONVEY_REVERSE :=, ENABLE_REVERSE := "+ST00330.RT01-PX1:4", ABS_ENABLE_FORWARD := "OPMODE01_DB".PowerOK.ST00325_RT01_VFD01, ABS_ENABLE_REVERSE := "OPMODE01_DB".PowerOK.ST00325_RT01_VFD01, FINE_POS_FORWARD :=, FINE_POS_REVERSE :=, POS_END_FORWARD_1 := "+ST00325.RT01-PX11:4", POS_END_FORWARD_2 :=, POS_END_REVERSE := "+ST00325.RT01-PX21:4", POS_SLOW_FORWARD := "+ST00325.RT01-PX12:4", POS_SLOW_REVERSE :=, POS_FOR_ACK := false, POS_REV_ACK :=, GAP_CONTROL_FORWARD :=, GAP_CONTROL_REVERSE :=, SELECT_FAST := #HMI_EXTENSION.Fast, "RUN_W/O_ENABLE" := #HMI_EXTENSION.Setup, DRIVE_READY := "ST00325_DB".RT01_VFD01.DRIVE_READY, DRIVE_RUNNING := "ST00325_DB".RT01_VFD01.DRIVE_RUNNING, EXTERNAL_ALARM := "ST00325_DB".Alarm, HIDE_ALARM_ALL := true, HIDE_ALARM_MASK :=, SET_OCC :=, RESET_OCC :=, OPMODE_USER_INTERFACE_OUT := "ST00325_DB".OPMODE, "GLOBAL_CLOCK&SYSTEM" := "GLOBAL_INFO_IDB".HMI_GLOBAL."Clock&System", IF_HMI := "GLOBAL_RT_2S2D1P_HMI_IF_DB".RT[25], IF_PARA_SET := "ST00325_DB".RT01.PARA_SET, HMI_SCREEN_AREA_POINTER := "GLOBAL_HMI_IF_DB".HMI_SCREEN_NO, HMI_SELECT_TIMESTAMP := "GLOBAL_HMI_IF_DB".HMI_SELECT_TIMESTAMP, FORWARD => "ST00325_DB".RT01.FORWARD, REVERSE => "ST00325_DB".RT01.REVERSE, FAST => "ST00325_DB".RT01.FAST, SLOW => "ST00325_DB".RT01.SLOW, JOG => "ST00325_DB".RT01.JOG, OPEN_BRAKE => "ST00325_DB".RT01.OPEN_BRAKE, GENERAL_ALARM => "ST00325_DB".RT01.GENERAL_ALARM, HS_TO_SUCCESSOR => "ST00325_DB".RT01.HS_TO_SUCCESSOR, HS_TO_PREDECESSOR => "ST00325_DB".RT01.HS_TO_PREDECESSOR, DISPLAY_OCCUPIED => "ST00325_DB".RT01.DISPLAY_OCCUPIED, DISPLAY_TRANSPORT => "ST00325_DB".RT01.DISPLAY_TRANSPORT, DISPLAY_IN_POSITION => "ST00325_DB".RT01.DISPLAY_IN_POSITION, DISPLAY_EMPTY => "ST00325_DB".RT01.DISPLAY_EMPTY, DISPLAY_OCCCARBODY => "ST00325_DB".RT01.DISPLAY_OCCCARBODY, DISPLAY_BLOCKENTRY => "ST00325_DB".RT01.DISPLAY_BLOCKENTRY, DISPLAY_BLOCKEXIT => "ST00325_DB".RT01.DISPLAY_BLOCKEXIT)
   END_RUNG
   RUNG wire#powerrail
      Contact( "ST00310_DB".VDL01.DISPLAY_INPOS1 )
      wire#w1
      Contact( "ST00325_DB".QRS01.READ_OK )
      wire#w2
      Contact( "ST00325_DB".SID01.DONE )
      { S7_Templates := "SrcType := DInt" } NE_Contact(in1 := "GLOBAL_RT_2S2D1P_HMI_IF_DB".RT[25].ActData.RTDataTarget, in2 := 0)
   END_RUNG wire#w3
   RUNG wire#w1
      Contact( "ST00325_SM_SA_FB_IDB".BYPASSED )
   END_RUNG wire#w2
   RUNG wire#powerrail
      Contact( "ST00310_DB".VDL01.DISPLAY_INPOS1 )
      Contact( "ST00310_DB".FX01.DISPLAY_POS_FORWARD )
   END_RUNG wire#w4
   RUNG wire#powerrail
      Contact( #HMI_EXTENSION.Forward )
   END_RUNG wire#w5
   RUNG wire#powerrail
      Contact( #HMI_EXTENSION.Backward )
   END_RUNG wire#w6
   // the same network as SCL:
   "ST00325_RT01_IDB"(PLANT_IDENTIFIER := WSTRING#'+ST00325.RT01',   // "RT_2S2D1P_PD_FB"
                      ENABLE_BLOCK := "CONTROL_ON_IDB".CONTROL_ON_DELAYED_1,
                      SAFETY_OK := "IF_SAFE_TO_STND_DB".OPMode01.SafetyOK.ST00325_RT01,
                      HS_FROM_SUCCESSOR := "ST00325_DB".HS_FROM_SUCCESSOR,
                      HS_FROM_PREDECESSOR := "ST00325_DB".HS_FROM_PREDECESSOR,
                      AUTO_CONVEY_FORWARD := "ST00310_DB".VDL01.DISPLAY_INPOS1 AND ("ST00325_DB".QRS01.READ_OK OR "ST00325_SM_SA_FB_IDB".BYPASSED) AND "ST00325_DB".SID01.DONE AND ("GLOBAL_RT_2S2D1P_HMI_IF_DB".RT[25].ActData.RTDataTarget <> 0),
                      ENABLE_FORWARD := "ST00310_DB".VDL01.DISPLAY_INPOS1 AND "ST00310_DB".FX01.DISPLAY_POS_FORWARD,
                      ENABLE_REVERSE := "+ST00330.RT01-PX1:4",
                      ABS_ENABLE_FORWARD := "OPMODE01_DB".PowerOK.ST00325_RT01_VFD01,
                      ABS_ENABLE_REVERSE := "OPMODE01_DB".PowerOK.ST00325_RT01_VFD01,
                      PB_FORWARD := #HMI_EXTENSION.Forward,
                      PB_REVERSE := #HMI_EXTENSION.Backward,
                      POS_END_FORWARD_1 := "+ST00325.RT01-PX11:4",
                      POS_END_REVERSE := "+ST00325.RT01-PX21:4",
                      POS_SLOW_FORWARD := "+ST00325.RT01-PX12:4",
                      POS_FOR_ACK := false,
                      SELECT_FAST := #HMI_EXTENSION.Fast,
                      "RUN_W/O_ENABLE" := #HMI_EXTENSION.Setup,
                      DRIVE_READY := "ST00325_DB".RT01_VFD01.DRIVE_READY,
                      DRIVE_RUNNING := "ST00325_DB".RT01_VFD01.DRIVE_RUNNING,
                      EXTERNAL_ALARM := "ST00325_DB".Alarm,
                      HIDE_ALARM_ALL := true,
                      OPMODE_USER_INTERFACE_OUT := "ST00325_DB".OPMODE,
                      "GLOBAL_CLOCK&SYSTEM" := "GLOBAL_INFO_IDB".HMI_GLOBAL."Clock&System",
                      IF_HMI := "GLOBAL_RT_2S2D1P_HMI_IF_DB".RT[25],
                      IF_PARA_SET := "ST00325_DB".RT01.PARA_SET,
                      HMI_SCREEN_AREA_POINTER := "GLOBAL_HMI_IF_DB".HMI_SCREEN_NO,
                      HMI_SELECT_TIMESTAMP := "GLOBAL_HMI_IF_DB".HMI_SELECT_TIMESTAMP,
                      FORWARD => "ST00325_DB".RT01.FORWARD,
                      REVERSE => "ST00325_DB".RT01.REVERSE,
                      FAST => "ST00325_DB".RT01.FAST,
                      SLOW => "ST00325_DB".RT01.SLOW,
                      JOG => "ST00325_DB".RT01.JOG,
                      OPEN_BRAKE => "ST00325_DB".RT01.OPEN_BRAKE,
                      GENERAL_ALARM => "ST00325_DB".RT01.GENERAL_ALARM,
                      HS_TO_SUCCESSOR => "ST00325_DB".RT01.HS_TO_SUCCESSOR,
                      HS_TO_PREDECESSOR => "ST00325_DB".RT01.HS_TO_PREDECESSOR,
                      DISPLAY_OCCUPIED => "ST00325_DB".RT01.DISPLAY_OCCUPIED,
                      DISPLAY_TRANSPORT => "ST00325_DB".RT01.DISPLAY_TRANSPORT,
                      DISPLAY_IN_POSITION => "ST00325_DB".RT01.DISPLAY_IN_POSITION,
                      DISPLAY_EMPTY => "ST00325_DB".RT01.DISPLAY_EMPTY,
                      DISPLAY_OCCCARBODY => "ST00325_DB".RT01.DISPLAY_OCCCARBODY,
                      DISPLAY_BLOCKENTRY => "ST00325_DB".RT01.DISPLAY_BLOCKENTRY,
                      DISPLAY_BLOCKEXIT => "ST00325_DB".RT01.DISPLAY_BLOCKEXIT);
END_REGION

REGION Network 34: RT01 Speed
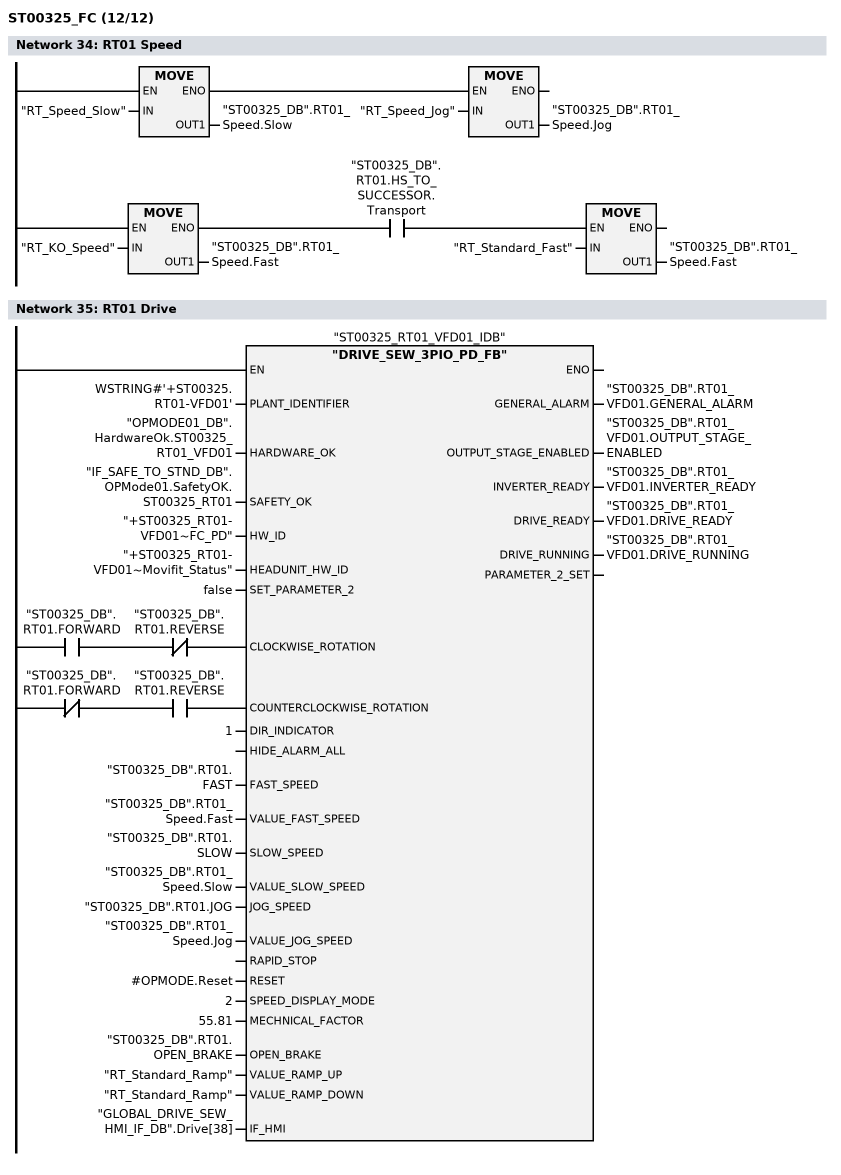
   RUNG wire#powerrail
      Move(in := "RT_Speed_Slow", out1 => "ST00325_DB".RT01_Speed.Slow)
      Move(in := "RT_Speed_Jog", out1 => "ST00325_DB".RT01_Speed.Jog)
   END_RUNG
   RUNG wire#powerrail
      Move(in := "RT_KO_Speed", out1 => "ST00325_DB".RT01_Speed.Fast)
      Contact( "ST00325_DB".RT01.HS_TO_SUCCESSOR.Transport )
      Move(in := "RT_Standard_Fast", out1 => "ST00325_DB".RT01_Speed.Fast)
   END_RUNG
   // the same network as SCL:
   "ST00325_DB".RT01_Speed.Slow := "RT_Speed_Slow";
   "ST00325_DB".RT01_Speed.Jog := "RT_Speed_Jog";
   "ST00325_DB".RT01_Speed.Fast := "RT_KO_Speed";
   IF "ST00325_DB".RT01.HS_TO_SUCCESSOR.Transport THEN
       "ST00325_DB".RT01_Speed.Fast := "RT_Standard_Fast";
   END_IF;
END_REGION

REGION Network 35: RT01 Drive
   RUNG wire#powerrail
      "ST00325_RT01_VFD01_IDB"(CLOCKWISE_ROTATION := wire#w1, COUNTERCLOCKWISE_ROTATION := wire#w2, PLANT_IDENTIFIER := WSTRING#'+ST00325.RT01-VFD01', HARDWARE_OK := "OPMODE01_DB".HardwareOk.ST00325_RT01_VFD01, SAFETY_OK := "IF_SAFE_TO_STND_DB".OPMode01.SafetyOK.ST00325_RT01, HW_ID := "+ST00325_RT01-VFD01~FC_PD", HEADUNIT_HW_ID := "+ST00325_RT01-VFD01~Movifit_Status", SET_PARAMETER_2 := false, DIR_INDICATOR := 1, HIDE_ALARM_ALL :=, FAST_SPEED := "ST00325_DB".RT01.FAST, VALUE_FAST_SPEED := "ST00325_DB".RT01_Speed.Fast, SLOW_SPEED := "ST00325_DB".RT01.SLOW, VALUE_SLOW_SPEED := "ST00325_DB".RT01_Speed.Slow, JOG_SPEED := "ST00325_DB".RT01.JOG, VALUE_JOG_SPEED := "ST00325_DB".RT01_Speed.Jog, RAPID_STOP :=, RESET := #OPMODE.Reset, SPEED_DISPLAY_MODE := 2, MECHNICAL_FACTOR := 55.81, OPEN_BRAKE := "ST00325_DB".RT01.OPEN_BRAKE, VALUE_RAMP_UP := "RT_Standard_Ramp", VALUE_RAMP_DOWN := "RT_Standard_Ramp", IF_HMI := "GLOBAL_DRIVE_SEW_HMI_IF_DB".Drive[38], GENERAL_ALARM => "ST00325_DB".RT01_VFD01.GENERAL_ALARM, OUTPUT_STAGE_ENABLED => "ST00325_DB".RT01_VFD01.OUTPUT_STAGE_ENABLED, INVERTER_READY => "ST00325_DB".RT01_VFD01.INVERTER_READY, DRIVE_READY => "ST00325_DB".RT01_VFD01.DRIVE_READY, DRIVE_RUNNING => "ST00325_DB".RT01_VFD01.DRIVE_RUNNING, PARAMETER_2_SET =>)
   END_RUNG
   RUNG wire#powerrail
      Contact( "ST00325_DB".RT01.FORWARD )
      I_Contact( "ST00325_DB".RT01.REVERSE )
   END_RUNG wire#w1
   RUNG wire#powerrail
      I_Contact( "ST00325_DB".RT01.FORWARD )
      Contact( "ST00325_DB".RT01.REVERSE )
   END_RUNG wire#w2
   // the same network as SCL:
   "ST00325_RT01_VFD01_IDB"(PLANT_IDENTIFIER := WSTRING#'+ST00325.RT01-VFD01',   // "DRIVE_SEW_3PIO_PD_FB"
                           HARDWARE_OK := "OPMODE01_DB".HardwareOk.ST00325_RT01_VFD01,
                           SAFETY_OK := "IF_SAFE_TO_STND_DB".OPMode01.SafetyOK.ST00325_RT01,
                           HW_ID := "+ST00325_RT01-VFD01~FC_PD",
                           HEADUNIT_HW_ID := "+ST00325_RT01-VFD01~Movifit_Status",
                           SET_PARAMETER_2 := false,
                           CLOCKWISE_ROTATION := "ST00325_DB".RT01.FORWARD AND NOT "ST00325_DB".RT01.REVERSE,
                           COUNTERCLOCKWISE_ROTATION := NOT "ST00325_DB".RT01.FORWARD AND "ST00325_DB".RT01.REVERSE,
                           DIR_INDICATOR := 1,
                           FAST_SPEED := "ST00325_DB".RT01.FAST,
                           VALUE_FAST_SPEED := "ST00325_DB".RT01_Speed.Fast,
                           SLOW_SPEED := "ST00325_DB".RT01.SLOW,
                           VALUE_SLOW_SPEED := "ST00325_DB".RT01_Speed.Slow,
                           JOG_SPEED := "ST00325_DB".RT01.JOG,
                           VALUE_JOG_SPEED := "ST00325_DB".RT01_Speed.Jog,
                           RESET := #OPMODE.Reset,
                           SPEED_DISPLAY_MODE := 2,
                           MECHNICAL_FACTOR := 55.81,
                           OPEN_BRAKE := "ST00325_DB".RT01.OPEN_BRAKE,
                           VALUE_RAMP_UP := "RT_Standard_Ramp",
                           VALUE_RAMP_DOWN := "RT_Standard_Ramp",
                           IF_HMI := "GLOBAL_DRIVE_SEW_HMI_IF_DB".Drive[38],
                           GENERAL_ALARM => "ST00325_DB".RT01_VFD01.GENERAL_ALARM,
                           OUTPUT_STAGE_ENABLED => "ST00325_DB".RT01_VFD01.OUTPUT_STAGE_ENABLED,
                           INVERTER_READY => "ST00325_DB".RT01_VFD01.INVERTER_READY,
                           DRIVE_READY => "ST00325_DB".RT01_VFD01.DRIVE_READY,
                           DRIVE_RUNNING => "ST00325_DB".RT01_VFD01.DRIVE_RUNNING);
END_REGION
END_FUNCTION
